(* CoDeSys 2.3.9.48 project: test.pro *)
(* Libraries: SysLibRtc.lib 8.11.10 11:37:48, SerComm.lib 31.5.11 08:06:48, C:\Stuff\Wago\libs\WagoLibDaylightSaving.lib 26.2.10 09:49:28, Building_common.lib 28.9.15 12:45:22, Standard.lib 8.11.10 11:37:48, C:\Stuff\Wago\libs\WagoBuilding_01.lib 21.3.16 16:30:58, WagoLibSSL.lib 25.2.13 12:47:14, SYSLIBCALLBACK.LIB 8.11.10 11:37:48, Ethernet.lib 8.11.10 11:37:48, C:\Stuff\Wago\libs\oscat_building_100.lib 2.1.18 20:06:49, C:\Stuff\Wago\libs\oscat_basic_333.lib 2.1.18 20:07:40 *)

(* PLC configuration (modules and I/O channels)
0750-1405 16 DI 24V DC 3.0ms [Type_1_16_Channels] node 0, in %IB0 out %QB0 {INTTypePAAssignment = PLC; INTTypeModule = plugged}
  in10 AT %IX0.0 [BOOLOnX_I] Ch_1 Digital input
  in11 AT %IX0.1 [BOOLOnX_I] Ch_2 Digital input
  in12 AT %IX0.2 [BOOLOnX_I] Ch_3 Digital input
  in13 AT %IX0.3 [BOOLOnX_I] Ch_4 Digital input
  in14 AT %IX0.4 [BOOLOnX_I] Ch_5 Digital input
  in15 AT %IX0.5 [BOOLOnX_I] Ch_6 Digital input
  in16 AT %IX0.6 [BOOLOnX_I] Ch_7 Digital input
  in17 AT %IX0.7 [BOOLOnX_I] Ch_8 Digital input
  in18 AT %IX0.8 [BOOLOnX_I] Ch_9 Digital input
  in19 AT %IX0.9 [BOOLOnX_I] Ch_10 Digital input
  in1A AT %IX0.10 [BOOLOnX_I] Ch_11 Digital input
  in1B AT %IX0.11 [BOOLOnX_I] Ch_12 Digital input
  in1C AT %IX0.12 [BOOLOnX_I] Ch_13 Digital input
  in1D AT %IX0.13 [BOOLOnX_I] Ch_14 Digital input
  in1E AT %IX0.14 [BOOLOnX_I] Ch_15 Digital input
  in1F AT %IX0.15 [BOOLOnX_I] Ch_16 Digital input
0750-0430 8 DI 24 V DC 3.0ms [Type_1_8_Channels] node 1, in %IB0 out %QB0 {INTTypePAAssignment = PLC; INTTypeModule = plugged}
  in20 AT %IX1.0 [BOOLOnX_I] Ch_1 Digital input
  in21 AT %IX1.1 [BOOLOnX_I] Ch_2 Digital input
  in22 AT %IX1.2 [BOOLOnX_I] Ch_3 Digital input
  in23 AT %IX1.3 [BOOLOnX_I] Ch_4 Digital input
  in24 AT %IX1.4 [BOOLOnX_I] Ch_5 Digital input
  in25 AT %IX1.5 [BOOLOnX_I] Ch_6 Digital input
  in26 AT %IX1.6 [BOOLOnX_I] Ch_7 Digital input
  in27 AT %IX1.7 [BOOLOnX_I] Ch_8 Digital input
0750-0430 8 DI 24 V DC 3.0ms [Type_1_8_Channels] node 2, in %IB2 out %QB0 {INTTypePAAssignment = PLC; INTTypeModule = plugged}
  in30 AT %IX1.8 [BOOLOnX_I] Ch_1 Digital input
  in31 AT %IX1.9 [BOOLOnX_I] Ch_2 Digital input
  in32 AT %IX1.10 [BOOLOnX_I] Ch_3 Digital input
  in33 AT %IX1.11 [BOOLOnX_I] Ch_4 Digital input
  in34 AT %IX1.12 [BOOLOnX_I] Ch_5 Digital input
  in35 AT %IX1.13 [BOOLOnX_I] Ch_6 Digital input
  in36 AT %IX1.14 [BOOLOnX_I] Ch_7 Digital input
  in37 AT %IX1.15 [BOOLOnX_I] Ch_8 Digital input
0750-0430 8 DI 24 V DC 3.0ms [Type_1_8_Channels] node 3, in %IB3 out %QB0 {INTTypePAAssignment = PLC; INTTypeModule = plugged}
  in40 AT %IX2.0 [BOOLOnX_I] Ch_1 Digital input
  in41 AT %IX2.1 [BOOLOnX_I] Ch_2 Digital input
  in42 AT %IX2.2 [BOOLOnX_I] Ch_3 Digital input
  in43 AT %IX2.3 [BOOLOnX_I] Ch_4 Digital input
  in44 AT %IX2.4 [BOOLOnX_I] Ch_5 Digital input
  in45 AT %IX2.5 [BOOLOnX_I] Ch_6 Digital input
  in46 AT %IX2.6 [BOOLOnX_I] Ch_7 Digital input
  in47 AT %IX2.7 [BOOLOnX_I] Ch_8 Digital input
0750-0402 4 DI 24 V DC 3.0ms [Type_1_4_Channels] node 4, in %IB4 out %QB0 {INTTypePAAssignment = PLC; INTTypeModule = plugged}
  in50 AT %IX2.8 [BOOLOnX_I] Ch_1 Digital input
  in51 AT %IX2.9 [BOOLOnX_I] Ch_2 Digital input
  in52 AT %IX2.10 [BOOLOnX_I] Ch_3 Digital input
  in53 AT %IX2.11 [BOOLOnX_I] Ch_4 Digital input
0750-0418 2 DI 24V DC 3.0ms / Diagnosis / Acknowledgement [Type_6_2_Channels] node 5, in %IB5 out %QB0 {INTTypePAAssignment = PLC; INTTypeModule = plugged}
  in60 AT %IX2.12 [BOOLOnX_I] Digital input
  in61 AT %IX2.13 [BOOLOnX_I] Digital input
  AT %IX2.14 [BOOLOnX_I] Diagnostic
  AT %IX2.15 [BOOLOnX_I] Diagnostic
  AT %QX0.2 [BOOLOnX_Q] Reset diagnostic
  AT %QX0.3 [BOOLOnX_Q] Reset diagnostic
0750-0418 2 DI 24V DC 3.0ms / Diagnosis / Acknowledgement [Type_6_2_Channels] node 6, in %IX2.12 out %QB0 {INTTypePAAssignment = PLC; INTTypeModule = plugged}
  in70 AT %IX3.0 [BOOLOnX_I] Digital input
  in71 AT %IX3.1 [BOOLOnX_I] Digital input
  AT %IX3.2 [BOOLOnX_I] Diagnostic
  AT %IX3.3 [BOOLOnX_I] Diagnostic
  AT %QX0.6 [BOOLOnX_Q] Reset diagnostic
  AT %QX0.7 [BOOLOnX_Q] Reset diagnostic
0750-0418 2 DI 24V DC 3.0ms / Diagnosis / Acknowledgement [Type_6_2_Channels] node 7, in %IB6 out %QX0.4 {INTTypePAAssignment = PLC; INTTypeModule = plugged}
  in80 AT %IX3.4 [BOOLOnX_I] Digital input
  in81 AT %IX3.5 [BOOLOnX_I] Digital input
  AT %IX3.6 [BOOLOnX_I] Diagnostic
  AT %IX3.7 [BOOLOnX_I] Diagnostic
  AT %QX0.10 [BOOLOnX_Q] Reset diagnostic
  AT %QX0.11 [BOOLOnX_Q] Reset diagnostic
0750-0418 2 DI 24V DC 3.0ms / Diagnosis / Acknowledgement [Type_6_2_Channels] node 8, in %IX3.4 out %QB1 {INTTypePAAssignment = PLC; INTTypeModule = plugged}
  in90 AT %IX3.8 [BOOLOnX_I] Digital input
  in91 AT %IX3.9 [BOOLOnX_I] Digital input
  AT %IX3.10 [BOOLOnX_I] Diagnostic
  AT %IX3.11 [BOOLOnX_I] Diagnostic
  AT %QX0.14 [BOOLOnX_Q] Reset diagnostic
  AT %QX0.15 [BOOLOnX_Q] Reset diagnostic
0750-0418 2 DI 24V DC 3.0ms / Diagnosis / Acknowledgement [Type_6_2_Channels] node 9, in %IB7 out %QX0.12 {INTTypePAAssignment = PLC; INTTypeModule = plugged}
  inA0 AT %IX3.12 [BOOLOnX_I] Digital input
  inA1 AT %IX3.13 [BOOLOnX_I] Digital input
  AT %IX3.14 [BOOLOnX_I] Diagnostic
  AT %IX3.15 [BOOLOnX_I] Diagnostic
  AT %QX1.2 [BOOLOnX_Q] Reset diagnostic
  AT %QX1.3 [BOOLOnX_Q] Reset diagnostic
0750-0418 2 DI 24V DC 3.0ms / Diagnosis / Acknowledgement [Type_6_2_Channels] node 10, in %IX3.12 out %QB2 {INTTypePAAssignment = PLC; INTTypeModule = plugged}
  inB0 AT %IX4.0 [BOOLOnX_I] Digital input
  inB1 AT %IX4.1 [BOOLOnX_I] Digital input
  AT %IX4.2 [BOOLOnX_I] Diagnostic
  AT %IX4.3 [BOOLOnX_I] Diagnostic
  AT %QX1.6 [BOOLOnX_Q] Reset diagnostic
  AT %QX1.7 [BOOLOnX_Q] Reset diagnostic
0750-0418 2 DI 24V DC 3.0ms / Diagnosis / Acknowledgement [Type_6_2_Channels] node 11, in %IB8 out %QX1.4 {INTTypePAAssignment = PLC; INTTypeModule = plugged}
  inC0 AT %IX4.4 [BOOLOnX_I] Digital input
  inC01 AT %IX4.5 [BOOLOnX_I] Digital input
  AT %IX4.6 [BOOLOnX_I] Diagnostic
  AT %IX4.7 [BOOLOnX_I] Diagnostic
  AT %QX1.10 [BOOLOnX_Q] Reset diagnostic
  AT %QX1.11 [BOOLOnX_Q] Reset diagnostic
0750-1504 16 DO 24V DC 0.5A [Type_10_16_Channels] node 12, in %IX4.4 out %QB3 {INTTypePAAssignment = PLC; INTTypeModule = plugged}
  out10 AT %QX1.12 [BOOLOnX_Q] Ch_1 Digital output
  out11 AT %QX1.13 [BOOLOnX_Q] Ch_2 Digital output
  out12 AT %QX1.14 [BOOLOnX_Q] Ch_3 Digital output
  out13 AT %QX1.15 [BOOLOnX_Q] Ch_4 Digital output
  out14 AT %QX2.0 [BOOLOnX_Q] Ch_5 Digital output
  out15 AT %QX2.1 [BOOLOnX_Q] Ch_6 Digital output
  out16 AT %QX2.2 [BOOLOnX_Q] Ch_7 Digital output
  out17 AT %QX2.3 [BOOLOnX_Q] Ch_8 Digital output
  out18 AT %QX2.4 [BOOLOnX_Q] Ch_9 Digital output
  out19 AT %QX2.5 [BOOLOnX_Q] Ch_10 Digital output
  out1A AT %QX2.6 [BOOLOnX_Q] Ch_11 Digital output
  out1B AT %QX2.7 [BOOLOnX_Q] Ch_12 Digital output
  out1C AT %QX2.8 [BOOLOnX_Q] Ch_13 Digital output
  out1D AT %QX2.9 [BOOLOnX_Q] Ch_14 Digital output
  out1E AT %QX2.10 [BOOLOnX_Q] Ch_15 Digital output
  out1F AT %QX2.11 [BOOLOnX_Q] Ch_16 Digital output
0750-1504 16 DO 24V DC 0.5A [Type_10_16_Channels] node 13, in %IB9 out %QX1.12 {INTTypePAAssignment = PLC; INTTypeModule = plugged}
  out20 AT %QX2.12 [BOOLOnX_Q] Ch_1 Digital output
  out21 AT %QX2.13 [BOOLOnX_Q] Ch_2 Digital output
  out22 AT %QX2.14 [BOOLOnX_Q] Ch_3 Digital output
  out23 AT %QX2.15 [BOOLOnX_Q] Ch_4 Digital output
  out24 AT %QX3.0 [BOOLOnX_Q] Ch_5 Digital output
  out25 AT %QX3.1 [BOOLOnX_Q] Ch_6 Digital output
  out26 AT %QX3.2 [BOOLOnX_Q] Ch_7 Digital output
  out27 AT %QX3.3 [BOOLOnX_Q] Ch_8 Digital output
  out28 AT %QX3.4 [BOOLOnX_Q] Ch_9 Digital output
  out29 AT %QX3.5 [BOOLOnX_Q] Ch_10 Digital output
  out2A AT %QX3.6 [BOOLOnX_Q] Ch_11 Digital output
  out2B AT %QX3.7 [BOOLOnX_Q] Ch_12 Digital output
  out2C AT %QX3.8 [BOOLOnX_Q] Ch_13 Digital output
  out2D AT %QX3.9 [BOOLOnX_Q] Ch_14 Digital output
  out2E AT %QX3.10 [BOOLOnX_Q] Ch_15 Digital output
  out2F AT %QX3.11 [BOOLOnX_Q] Ch_16 Digital output
0750-1504 16 DO 24V DC 0.5A [Type_10_16_Channels] node 14, in %IB9 out %QX2.12 {INTTypePAAssignment = PLC; INTTypeModule = plugged}
  out30 AT %QX3.12 [BOOLOnX_Q] Ch_1 Digital output
  out31 AT %QX3.13 [BOOLOnX_Q] Ch_2 Digital output
  out32 AT %QX3.14 [BOOLOnX_Q] Ch_3 Digital output
  out33 AT %QX3.15 [BOOLOnX_Q] Ch_4 Digital output
  out34 AT %QX4.0 [BOOLOnX_Q] Ch_5 Digital output
  out35 AT %QX4.1 [BOOLOnX_Q] Ch_6 Digital output
  out36 AT %QX4.2 [BOOLOnX_Q] Ch_7 Digital output
  out37 AT %QX4.3 [BOOLOnX_Q] Ch_8 Digital output
  out38 AT %QX4.4 [BOOLOnX_Q] Ch_9 Digital output
  out39 AT %QX4.5 [BOOLOnX_Q] Ch_10 Digital output
  out3A AT %QX4.6 [BOOLOnX_Q] Ch_11 Digital output
  out3B AT %QX4.7 [BOOLOnX_Q] Ch_12 Digital output
  out3C AT %QX4.8 [BOOLOnX_Q] Ch_13 Digital output
  out3D AT %QX4.9 [BOOLOnX_Q] Ch_14 Digital output
  out3E AT %QX4.10 [BOOLOnX_Q] Ch_15 Digital output
  out3F AT %QX4.11 [BOOLOnX_Q] Ch_16 Digital output
0750-0517 2 DO 230V AC 1.0A Rel 2CO (PotFree) [Type_10_2_Channels] node 15, in %IB9 out %QX3.12 {INTTypePAAssignment = PLC; INTTypeModule = plugged}
  out40 AT %QX4.12 [BOOLOnX_Q] Ch_1 Digital output
  out41 AT %QX4.13 [BOOLOnX_Q] Ch_2 Digital output
0750-0517 2 DO 230V AC 1.0A Rel 2CO (PotFree) [Type_10_2_Channels] node 16, in %IB9 out %QX4.12 {INTTypePAAssignment = PLC; INTTypeModule = plugged}
  out50 AT %QX4.14 [BOOLOnX_Q] Ch_1 Digital output
  out51 AT %QX4.15 [BOOLOnX_Q] Ch_2 Digital output
0750-0517 2 DO 230V AC 1.0A Rel 2CO (PotFree) [Type_10_2_Channels] node 17, in %IB9 out %QX4.14 {INTTypePAAssignment = PLC; INTTypeModule = plugged}
  out60 AT %QX5.0 [BOOLOnX_Q] Ch_1 Digital output
  out61 AT %QX5.1 [BOOLOnX_Q] Ch_2 Digital output
0750-0517 2 DO 230V AC 1.0A Rel 2CO (PotFree) [Type_10_2_Channels] node 18, in %IB9 out %QB10 {INTTypePAAssignment = PLC; INTTypeModule = plugged}
  out70 AT %QX5.2 [BOOLOnX_Q] Ch_1 Digital output
  out71 AT %QX5.3 [BOOLOnX_Q] Ch_2 Digital output
0750-0513 2 DO 250V AC 2.0A Rel 2NO (PotFree) [Type_10_2_Channels] node 19, in %IB9 out %QX5.2 {INTTypePAAssignment = PLC; INTTypeModule = plugged}
  out80 AT %QX5.4 [BOOLOnX_Q] Ch_1 Digital output
  out81 AT %QX5.5 [BOOLOnX_Q] Ch_2 Digital output
AT %IX4.8 [BOOLOnX_I] Channel 1 Diagnostic bit 0
AT %IX4.9 [BOOLOnX_I] Channel 1 Diagnostic bit 1
AT %IX4.10 [BOOLOnX_I] Channel 2 Diagnostic bit 0
AT %IX4.11 [BOOLOnX_I] Channel 2 Diagnostic bit 1
out90 AT %QX5.6 [BOOLOnX_Q] Digital output 1
out91 AT %QX5.7 [BOOLOnX_Q] Digital output 2
AT %IX4.12 [BOOLOnX_I] Channel 1 Diagnostic bit 0
AT %IX4.13 [BOOLOnX_I] Channel 1 Diagnostic bit 1
AT %IX4.14 [BOOLOnX_I] Channel 2 Diagnostic bit 0
AT %IX4.15 [BOOLOnX_I] Channel 2 Diagnostic bit 1
outA0 AT %QX5.10 [BOOLOnX_Q] Digital output 1
out1A1 AT %QX5.11 [BOOLOnX_Q] Digital output 2
AT %IX5.0 [BOOLOnX_I] Channel 1 Diagnostic bit 0
AT %IX5.1 [BOOLOnX_I] Channel 1 Diagnostic bit 1
AT %IX5.2 [BOOLOnX_I] Channel 2 Diagnostic bit 0
AT %IX5.3 [BOOLOnX_I] Channel 2 Diagnostic bit 1
outB0 AT %QX5.14 [BOOLOnX_Q] Digital output 1
outB1 AT %QX5.15 [BOOLOnX_Q] Digital output 2
Fieldbus variables [FB_VARS] node 1, in %IB0 out %QB0
Flag variables [FLAG_VARS] node 2, in %IB0 out %QB0
Modbus-Master [MB_MASTER] node 3, in %IB0 out %QB0
*)

(* Task configuration *)
TASK MainTask (PRIORITY := 1); (* freewheeling *)
	PLC_PRG();
END_TASK
TASK UpdateClock (PRIORITY := 3, INTERVAL := T#1000ms);
	ReadClock();
END_TASK

(* POU PLC_PRG, ST *)
PROGRAM PLC_PRG
VAR
	pompaCWU:FbLatchedRelay;
	pompaCWUVis:BOOL;
	pompaCWUTOF:TOF;
	pompaCWUTOFTRIG:F_TRIG;

	tvSat:FbLatchedRelay;
	tvSatVis:BOOL;
	tvSatTOF:TOF;
	tvSatTOFTRIG:F_TRIG;
END_VAR
Swiatlo;
SterowanieRolet;

pompaCWU(xButton:=(LazienkaPietro.Swiatlo OR LazienkaParter.Swiatlo OR KuchniaJadalnia.Swiatlo OR pompaCWUVis), xCentralOff:=pompaCWUTOFTRIG.Q);
pompaCWUTOF(IN:=LazienkaPietro.swLazienkaD.xActuator,PT:=T#10M);
pompaCWUTOFTRIG(CLK:=pompaCWUTOF.Q);
out2C:=pompaCWU.xActuator;

(*TODOultimate off*)

(*TVSAT off*)
END_PROGRAM

(* POU Swiatlo, ST *)
PROGRAM Swiatlo
VAR

END_VAR
GarazKotlownia;
GarderobaStrych;
Korytarz;
KuchniaJadalnia;
LazienkaParter;
LazienkaPietro;
PokojPolnoc;
PokojPoludnie;
Salon;
Sypialnia;
WiatrolapSpizarnia;
END_PROGRAM

(* POU Swiatlo2/GarazKotlownia, ST *)
PROGRAM GarazKotlownia
VAR
	swGarazDrzwiKotlowni : BOOL;
	visGaraz : BOOL;
	swGarazBrama: BOOL;
	swGarazBiurko: BOOL;
	garazTOF:TOF;
	garazTOFTRIG:F_TRIG;
	garazClicker: CLICK;
	wlaczWszystkieSw: BOOL := FALSE;
	wylaczWszystkieSw: BOOL := FALSE;
	visKotlownia: BOOL;
	kotlowniaTOF:TOF;
	kotlowniaTOFTRIG:F_TRIG;
	kotlowniaClicker: FbWB_EvaluateMultipleClicks;
	garaz:SwiatloOpFUN;
END_VAR
VAR RETAIN
	swGaraz: FbLatchedRelay;
	swKotlownia: FbLatchedRelay;
END_VAR
(*----------Garaz--------*)
(*swGaraz(xButton:= (garazClicker.single OR garazClicker.double OR visGaraz), xCentralOn:=wlaczWszystkieSw, xCentralOff:=garazTOFTRIG.Q);
out10:=swGaraz.xActuator;
garazTOF(IN:=garazClicker.single, PT:=T#2M);
garazTOFTRIG(CLK:=garazTOF.Q);
garazClicker(in:=(in10 OR in20));*)

garaz(wejscieSterujace:=(in10),wlaczWszystkie:=wlaczWszystkieSw,wylaczWszystkie:=wylaczWszystkieSw,sterowanieVis:=visGaraz);
out10:=garaz.wyjscie;

(*----------Kotlownia-------*)
swKotlownia(xButton:=(kotlowniaClicker.xMultipleClick OR kotlowniaClicker.xFewerClick OR visKotlownia), xCentralOn:=wlaczWszystkieSw, xCentralOff:=kotlowniaTOFTRIG.Q);
kotlowniaTOF(IN:=kotlowniaClicker.xFewerClick,PT:=T#5M);
kotlowniaTOFTRIG(CLK:=kotlowniaTOF.Q);
kotlowniaClicker(xButton:=(in11 OR in21));
out11:=swKotlownia.xActuator;
out90:=garaz.wyjscie;
out91:=garaz.wyjscie;
outA0:=garaz.wyjscie;
out1A1:=garaz.wyjscie;
outB0:=garaz.wyjscie;
outB1:=garaz.wyjscie;
END_PROGRAM

(* POU Swiatlo2/SwiatloOpFUN, ST *)
FUNCTION_BLOCK SwiatloOpFUN
VAR_INPUT
	wejscieSterujace :BOOL;
	wlaczWszystkie:BOOL;
	wylaczWszystkie:BOOL;
	sterowanieVis:BOOL;
END_VAR
VAR_OUTPUT
	wyjscie :BOOL;
END_VAR
VAR
	przelacznik:FbLatchedRelay;
	opoznienieTOF:TOF;
	opoznienieTOFTRIG:F_TRIG;
	clicker:Fb_Click;
END_VAR
przelacznik(xButton:=(clicker.xSingle OR clicker.xDouble OR  sterowanieVis), xCentralOn:=wlaczWszystkie, xCentralOff:=(opoznienieTOFTRIG.Q OR wylaczWszystkie));
opoznienieTOF(IN:=clicker.xSingle, PT:=T#3m);
opoznienieTOFTRIG(CLK:=opoznienieTOF.Q);
clicker(xSwitch:=wejscieSterujace,uiT_10tel_s:=5);
wyjscie:=przelacznik.xActuator;
END_FUNCTION_BLOCK

(* POU Swiatlo2/GarderobaStrych, ST *)
PROGRAM GarderobaStrych
VAR
	swStrych: FbLatchedRelay;
	visStrych: BOOL;
	strychTOF:TOF;
	strychTOFTRIG:F_TRIG;
	strychClicker: FbWB_EvaluateMultipleClicks;
	swSchowekPietro: FbLatchedRelay;
	visSchowekPietro: BOOL;
	schowekPietroTOF:TOF;
	schowekPietroTOFTRIG:F_TRIG;
	schowekPietroClicker: FbWB_EvaluateMultipleClicks;
	wlaczWszystkieSw: BOOL:=FALSE;
	wylaczWszystkieSw: BOOL:=FALSE;
END_VAR
swSchowekPietro(xButton:=(schowekPietroClicker.xMultipleClick OR schowekPietroClicker.xFewerClick OR visSchowekPietro),xCentralOn:=wlaczWszystkieSw,xCentralOff:=schowekPietroTOFTRIG.Q);
out25:=swSchowekPietro.xActuator;
schowekPietroTOF(IN:=schowekPietroClicker.xFewerClick,PT:=T#2m);
schowekPietroTOFTRIG(CLK:=schowekPietroTOF.Q);
schowekPietroClicker(xButton:=in34,bNumberOfClicks:=2);

swStrych(xButton:=(strychClicker.xMultipleClick OR strychTOFTRIG.Q OR visStrych), xCentralOn:=wlaczWszystkieSw,xCentralOff:=strychTOFTRIG.Q);
out26:=swStrych.xActuator;
strychTOF(IN:=strychClicker.xFewerClick,PT:=T#10m);
strychTOFTRIG(CLK:=strychTOF.Q);
strychClicker(xButton:=in35,bNumberOfClicks:=2);
END_PROGRAM

(* POU Swiatlo2/Korytarz, ST *)
PROGRAM Korytarz
VAR
	swKorytarz: FbLatchedRelay;
	visKorytarz: BOOL;
	swKorytarzPietro: FbLatchedRelay;
	visKorytarzPietro: BOOL;
	wlaczWszystkieSw: BOOL:=FALSE;
	wylaczWszystkieSw: BOOL:=FALSE;
END_VAR
swKorytarz(xButton:=(in1D OR visKorytarz), xCentralOn:=wlaczWszystkieSw, xCentralOff:=wylaczWszystkieSw);
out1D:=swKorytarz.xActuator;

swKorytarzPietro(xButton:=(in1F OR visKorytarzPietro), xCentralOn:=wlaczWszystkieSw, xCentralOff:=wylaczWszystkieSw);
out1F:=swKorytarzPietro.xActuator;
END_PROGRAM

(* POU Swiatlo2/KuchniaJadalnia, ST *)
PROGRAM KuchniaJadalnia
VAR
	swJadalnia: FbLatchedRelay;
	visJadalnia: BOOL;
	swBlat: FbLatchedRelay;
	visBlat: BOOL;
	swMeble: FbLatchedRelay;
	visMeble: BOOL;
	wlaczWszystkieSw: BOOL:=FALSE;
	wylaczWszystkieSw: BOOL:=FALSE;
	swSufit: FbLatchedRelay;
	visSufit: BOOL;
	swiatlo:BOOL;
END_VAR
(*----------Kuchnia--------------*)
swBlat(xButton:=(in17 OR visBlat), xCentralOn:=wlaczWszystkieSw,  xCentralOff:=wylaczWszystkieSw);
out16:=swBlat.xActuator;
swMeble(xButton:=(in16 OR visMeble), xCentralOn:=wlaczWszystkieSw,  xCentralOff:=wylaczWszystkieSw);
out17:=swMeble.xActuator;
swSufit(xButton:=(in16 OR visSufit), xCentralOn:=wlaczWszystkieSw,  xCentralOff:=wylaczWszystkieSw);
out1E:=swSufit.xActuator;

(*----------Jadalnia--------------*)
swJadalnia(xButton:=(in18 OR visJadalnia), xCentralOn:=wlaczWszystkieSw,xCentralOff:=wylaczWszystkieSw);
out18:=swJadalnia.xActuator;

Swiatlo:=swBlat.xActuator OR swMeble.xActuator OR swSufit.xActuator;
END_PROGRAM

(* POU Swiatlo2/LazienkaParter, ST *)
PROGRAM LazienkaParter
VAR
	visMalaLazienkaPrysznic:BOOL;
	swMalaLazienkaLustro: FbLatchedRelay;
	visMalaLazienkaLustro: BOOL;
	swMalaLazienka: FbLatchedRelay;
	visMalaLazienka: BOOL;
	swMalaLazienkaPrysznic: FbLatchedRelay;
	wlaczWszystkieSw: BOOL:=FALSE;
	wylaczWszystkieSw: BOOL:=FALSE;
	swiatlo: BOOL;
END_VAR
(*---------Mala lazienka -------*)
swMalaLazienka(xButton:=(in13 OR visMalaLazienka), xCentralOn:=wlaczWszystkieSw, xCentralOff:=wylaczWszystkieSw);
out13:=swMalaLazienka.xActuator;
swMalaLazienkaPrysznic(xButton:=(in14 OR in24 OR visMalaLazienkaPrysznic), xCentralOn:=wlaczWszystkieSw, xCentralOff:=wylaczWszystkieSw);
out50:=swMalaLazienkaPrysznic.xActuator;
swMalaLazienkaLustro(xButton:=(in15 OR in25 OR visMalaLazienkaLustro), xCentralOn:=wlaczWszystkieSw,xCentralOff:=wylaczWszystkieSw);
out15:=swMalaLazienkaLustro.xActuator;

Swiatlo:=swMalaLazienka.xActuator OR swMalaLazienkaPrysznic.xActuator OR swMalaLazienkaLustro.xActuator;
END_PROGRAM

(* POU Swiatlo2/LazienkaPietro, ST *)
PROGRAM LazienkaPietro
VAR
	swLustroLD: FbLatchedRelay;
	visLustroLD: BOOL;
	swLazienkaD: FbLatchedRelay;
	visLazienkaD: BOOL;
	swBlatLD: FbLatchedRelay;
	visBlatLD: BOOL;
	swPrysznicLD: FbLatchedRelay;
	visPrysznicLD: BOOL;

	swLazienkaLedTrigger: R_TRIG;
	visLedLD: BOOL;
	wlaczWszystkieSw: BOOL:=FALSE;
	wylaczWszystkieSw: BOOL:=FALSE;
	swiatlo:BOOL;
END_VAR
(*----------------Duza lazienka------------*)
swLustroLD(xButton:=(in36 OR visLustroLD), xCentralOn:=wlaczWszystkieSw,xCentralOff:=wylaczWszystkieSw);
out27:=swLustroLD.xActuator;
swLazienkaD(xButton:=(in37 OR visLazienkaD), xCentralOn:=wlaczWszystkieSw,xCentralOff:=wylaczWszystkieSw);
out28:=swLazienkaD.xActuator;
swBlatLD(xButton:=(in40 OR visBlatLD), xCentralOn:=wlaczWszystkieSw,xCentralOff:=wylaczWszystkieSw);
out40:=swBlatLD.xActuator;
swPrysznicLD(xButton:=(in41 OR visPrysznicLD), xCentralOn:=wlaczWszystkieSw,xCentralOff:=wylaczWszystkieSw);
out41:=swPrysznicLD.xActuator;

swLazienkaLedTrigger(CLK:=(in43 OR visLedLD));
IF swLazienkaLedTrigger.Q THEN
	IF NOT (out29 OR out2A) THEN
		visBlatLD := visPrysznicLD := TRUE;
	ELSE
		visBlatLD := visPrysznicLD := FALSE;
	END_IF;
END_IF;

Swiatlo:=swLazienkaD.xActuator OR swLustroLD.xActuator OR swBlatLD.xActuator OR swPrysznicLD.xActuator;
END_PROGRAM

(* POU Swiatlo2/PokojPolnoc, ST *)
PROGRAM PokojPolnoc
VAR
	swPokojPolnoc: FbLatchedRelay;
	visPokojPolnoc: BOOL;
	wlaczWszystkieSw: BOOL:=FALSE;
	wylaczWszystkieSw: BOOL:=FALSE;
END_VAR
swPokojPolnoc(xButton:=(in33 OR visPokojPolnoc),xCentralOn:=wlaczWszystkieSw,xCentralOff:=wylaczWszystkieSw);
out24:=swPokojPolnoc.xActuator;
END_PROGRAM

(* POU Swiatlo2/PokojPoludnie, ST *)
PROGRAM PokojPoludnie
VAR
	swPokojPoludnie: FbLatchedRelay;
	visPokojPoludnie: BOOL;
	wlaczWszystkieSw: BOOL:=FALSE;
	wylaczWszystkieSw: BOOL:=FALSE;
END_VAR
swPokojPoludnie(xButton:=(in32 OR visPokojPoludnie), xCentralOn:=wlaczWszystkieSw,xCentralOff:=wylaczWszystkieSw);
out23:=swPokojPoludnie.xActuator;
END_PROGRAM

(* POU Swiatlo2/Salon, ST *)
PROGRAM Salon
VAR
	swSalonCentralne: FbLatchedRelay;
	visSalonCentralne: BOOL;
	swSalonSciana: FbLatchedRelay;
	visSalonSciana: BOOL;
	swSalonKinkiet: FbLatchedRelay;
	visSalonKinkiet: BOOL;
	swSalonSufit: FbLatchedRelay;
	visSalonSufit: BOOL;
	wlaczWszystkieSw: BOOL:=FALSE;
	wylaczWszystkieSw: BOOL:=FALSE;
END_VAR
(*----------Salon-----------------*)
swSalonCentralne(xButton:=(in19 OR visSalonCentralne), xCentralOn:=wlaczWszystkieSw, xCentralOff:=wylaczWszystkieSw);
out19:=swSalonCentralne.xActuator;
swSalonSciana(xButton:=(in1A OR visSalonSciana), xCentralOn:=wlaczWszystkieSw, xCentralOff:=wylaczWszystkieSw);
out1A:=swSalonSciana.xActuator;
swSalonKinkiet(xButton:=(in1B OR visSalonKinkiet), xCentralOn:=wlaczWszystkieSw, xCentralOff:=wylaczWszystkieSw);
out1B:=swSalonKinkiet.xActuator;
swSalonSufit(xButton:=(in1C OR visSalonSufit), xCentralOn:=wlaczWszystkieSw, xCentralOff:=wylaczWszystkieSw);
out1C:=swSalonSufit.xActuator;
END_PROGRAM

(* POU Swiatlo2/Sypialnia, ST *)
PROGRAM Sypialnia
VAR
	swSypialniaLozko: FbLatchedRelay;
	visSypialniaLozko: BOOL;
	swSypialnia: FbLatchedRelay;
	visSypialnia: BOOL;
	wlaczWszystkieSw: BOOL:=FALSE;
	wylaczWszystkieSw: BOOL:=FALSE;
END_VAR
swSypialniaLozko(xButton:=(in26 OR visSypialniaLozko), xCentralOn:=wlaczWszystkieSw, xCentralOff:=wylaczWszystkieSw);
out20:=swSypialniaLozko.xActuator;

swSypialnia(xButton:=(in27 OR visSypialnia), xCentralOn:=wlaczWszystkieSw, xCentralOff:=wylaczWszystkieSw);
out21:=swSypialnia.xActuator;
END_PROGRAM

(* POU Swiatlo2/WiatrolapSpizarnia, ST *)
PROGRAM WiatrolapSpizarnia
VAR
	swWiatrolap:FbLatchedRelay;
	visWiatrolap:BOOL;
	wiatrolapTOF:TOF;
	wiatrolapTOFTRIG:F_TRIG;
	wiatrolapClicker:CLICK;
	wlaczWszystkieSw: BOOL:=FALSE;
	wylaczWszystkieSw: BOOL:=FALSE;
	swSpizarnia:SwiatloOpFUN;
	visSpizarnia:BOOL;
END_VAR
(*---------Wiatrolap--------*)
swWiatrolap(xButton:=(in12), xCentralOn:=wlaczWszystkieSw, xCentralOff:=wiatrolapTOFTRIG.Q);
wiatrolapTOF(IN:=wiatrolapClicker.single, PT:=T#5m);
wiatrolapTOFTRIG(CLK:=wiatrolapTOF.Q);
wiatrolapClicker(in:=in12);
out12:=swWiatrolap.xActuator;

(*-----Spizarnia---------*)
swSpizarnia(wejscieSterujace:=in1E,
	wlaczWszystkie:=wlaczWszystkieSw,
	wylaczWszystkie:=wylaczWszystkieSw,
	sterowanieVis:=visSpizarnia);
out14:=swSpizarnia.wyjscie;
END_PROGRAM

(* POU Rolety2/SterowanieRolet, ST *)
PROGRAM SterowanieRolet
VAR
	kotlownia: RoletyFUN;
	kotlowniaUpVis: BOOL;
	kotlowniaDnVis: BOOL;
	kotlowniaLamelkiVis: BOOL;

	witrynaP:RoletyFUN;
	witrynaL:RoletyFUN;
	witrynaUpVis:BOOL;
	witrynaDnVis:BOOL;
	witrynaLamelkiVis:BOOL;

	salonWyjscie: RoletyFUN;
	salonWyjscieUpVis:BOOL;
	salonWyjscieDnVis:BOOL;
	salonWyjscieLamelkiVis:BOOL;

	jadalniaWyjscie: RoletyFUN;
	jadalniaWyjscieUpVis:BOOL;
	jadalniaWyjscieDnVis:BOOL;
	jadalniaWyjscieLamelkiVis:BOOL;

	jadalniaWitryna: RoletyFUN;
	jadalniaWitrynaUpVis:BOOL;
	jadalniaWitrynaDnVis:BOOL;
	jadalniaWitrynaLamelkiVis:BOOL;

	kuchnia: RoletyFUN;
	kuchniaUpVis:BOOL;
	kuchniaDnVis:BOOL;
	kuchniaLamelkiVis:BOOL;

	lazienkaParterR: RoletyFUN;
	lazienkaParterUpVis:BOOL;
	lazienkaParterDnVis:BOOL;
	lazienkaParterLamelkiVis:BOOL;

	lazienkaPietroR: RoletyFUN;
	lazienkaPietroUpVis:BOOL;
	lazienkaPietroDnVis:BOOL;
	lazienkaPietroLamelkiVis:BOOL;

	pokojPolnocR: RoletyFUN;
	pokojPolnocUpVis:BOOL;
	pokojPolnocDnVis:BOOL;
	pokojPolnocLamelkiVis:BOOL;

	pokojPoludnieR: RoletyFUN;
	pokojPoludnieUpVis:BOOL;
	pokojPoludnieDnVis:BOOL;
	pokojPoludnieLamelkiVis:BOOL;

	sypialniaR: RoletyFUN;
	sypialniaUpVis:BOOL;
	sypialniaDnVis:BOOL;
	sypialniaLamelkiVis:BOOL;

	sypialniaBalkonR: RoletyFUN;
	sypialniaBalkonUpVis:BOOL;
	sypialniaBalkonDnVis:BOOL;
	sypialniaBalkonLamelkiVis:BOOL;

	zamykanieWszystkieVis: BOOL;
	otwieranieWszystkieVis: BOOL;
	podniesStrefeDzienna:BOOL;
	opuscStrefeDzienna:BOOL;
	podniesPietro:BOOL;
	opuscPietro:BOOL;
       roletyParter : Fb_ShortLong:=(uiTS_10tel_s:=1, uiTL_10tel_s:=1, uiT_10tel_s :=5);
	roletyPietro : Fb_ShortLong:=(uiTS_10tel_s:=1, uiTL_10tel_s:=1, uiT_10tel_s :=5);
	roletyParterPoludnie:Fb_ShortLong:=(uiTS_10tel_s:=1, uiTL_10tel_s:=1, uiT_10tel_s :=5);
	roletyParterPolnoc:Fb_ShortLong:=(uiTS_10tel_s:=1, uiTL_10tel_s:=1, uiT_10tel_s :=5);
	opuscParterPoludnie:BOOL;
	podniesParterPoludnie:BOOL;
	opuscParterPolnoc:BOOL;
	podniesParterPolnoc:BOOL;
END_VAR
roletyParter(xSwitch:=inC0);
roletyPietro(xSwitch:=inC01);
roletyParterPoludnie(xSwitch:=in20);
roletyParterPolnoc(xSwitch:=in23);
podniesStrefeDzienna:=roletyParter.xShort;
opuscStrefeDzienna:=roletyParter.xLong;
podniesPietro:=roletyPietro.xShort;
opuscPietro:=roletyPietro.xLong;
opuscParterPoludnie:=roletyParterPoludnie.xLong;
podniesParterPoludnie:=roletyParterPoludnie.xShort;
opuscParterPolnoc:=roletyParterPolnoc.xLong;
podniesParterPolnoc:=roletyParterPolnoc.xShort;

kotlownia(wejscieSterujace:=in60,
		ZmiennaPodnoszenieVis:=kotlowniaUpVis,
		ZmiennaOpuszczanieVis:=kotlowniaDnVis,
		ZmiennaLamelkiVis:=kotlowniaLamelkiVis,
		PozycjaLameli:=10,
		CzasOtwarcia:=T#15s,
		CzasZamkniecia:=T#13s,
		MaxCzasDzialania:=T#20s,
		ZamykanieWszystkieVis:=zamykanieWszystkieVis,
		OtwieranieWszystkieVis:=otwieranieWszystkieVis);
out51:=kotlownia.WyjsciePodnoszenie;
out60:=kotlownia.WyjscieOpuszczanie;

witrynaP(wejscieSterujace:=in61,
		ZmiennaPodnoszenieVis:=witrynaUpVis,
		ZmiennaOpuszczanieVis:=witrynaDnVis,
		ZmiennaLamelkiVis:=witrynaLamelkiVis,
		PozycjaLameli:=10,
		CzasOtwarcia:=T#30s,
		CzasZamkniecia:=T#25s,
		MaxCzasDzialania:=T#30s,
		ZamykanieWszystkieVis:=zamykanieWszystkieVis OR opuscStrefeDzienna OR opuscParterPoludnie,
		OtwieranieWszystkieVis:=otwieranieWszystkieVis OR podniesStrefeDzienna OR podniesParterPoludnie);
out61:=witrynaP.WyjsciePodnoszenie;
out70:=witrynaP.WyjscieOpuszczanie;

witrynaL(wejscieSterujace:=in61,
		ZmiennaPodnoszenieVis:=witrynaUpVis,
		ZmiennaOpuszczanieVis:=witrynaDnVis,
		ZmiennaLamelkiVis:=witrynaLamelkiVis,
		PozycjaLameli:=10,
		CzasOtwarcia:=T#30s,
		CzasZamkniecia:=T#25s,
		MaxCzasDzialania:=T#30s,
		ZamykanieWszystkieVis:=zamykanieWszystkieVis OR opuscStrefeDzienna OR opuscParterPoludnie,
		OtwieranieWszystkieVis:=otwieranieWszystkieVis OR podniesStrefeDzienna OR podniesParterPoludnie);
out71:=witrynaL.WyjsciePodnoszenie;
out80:=witrynaL.WyjscieOpuszczanie;

salonWyjscie(wejscieSterujace:=in70,
		ZmiennaPodnoszenieVis:=salonWyjscieUpVis,
		ZmiennaOpuszczanieVis:=salonWyjscieDnVis,
		ZmiennaLamelkiVis:=salonWyjscieLamelkiVis,
		PozycjaLameli:=10,
		CzasOtwarcia:=T#30s,
		CzasZamkniecia:=T#25s,
		MaxCzasDzialania:=T#30s,
		ZamykanieWszystkieVis:=zamykanieWszystkieVis OR opuscStrefeDzienna OR opuscParterPoludnie,
		OtwieranieWszystkieVis:=otwieranieWszystkieVis OR podniesStrefeDzienna OR podniesParterPoludnie);
out31:=salonWyjscie.WyjsciePodnoszenie;
out32:=salonWyjscie.WyjscieOpuszczanie;

jadalniaWyjscie(wejscieSterujace:=in71,
		ZmiennaPodnoszenieVis:=jadalniaWyjscieUpVis,
		ZmiennaOpuszczanieVis:=jadalniaWyjscieDnVis,
		ZmiennaLamelkiVis:=jadalniaWyjscieLamelkiVis,
		PozycjaLameli:=10,
		CzasOtwarcia:=T#30s,
		CzasZamkniecia:=T#25s,
		MaxCzasDzialania:=T#30s,
		ZamykanieWszystkieVis:=zamykanieWszystkieVis OR opuscStrefeDzienna OR opuscParterPolnoc,
		OtwieranieWszystkieVis:=otwieranieWszystkieVis OR podniesStrefeDzienna OR podniesParterPolnoc);
out33:=jadalniaWyjscie.WyjsciePodnoszenie;
out34:=jadalniaWyjscie.WyjscieOpuszczanie;

jadalniaWitryna(wejscieSterujace:=in80,
		ZmiennaPodnoszenieVis:=jadalniaWitrynaUpVis,
		ZmiennaOpuszczanieVis:=jadalniaWitrynaDnVis,
		ZmiennaLamelkiVis:=jadalniaWitrynaLamelkiVis,
		PozycjaLameli:=10,
		CzasOtwarcia:=T#30s,
		CzasZamkniecia:=T#25s,
		MaxCzasDzialania:=T#30s,
		ZamykanieWszystkieVis:=zamykanieWszystkieVis OR opuscStrefeDzienna OR opuscParterPolnoc,
		OtwieranieWszystkieVis:=otwieranieWszystkieVis OR podniesStrefeDzienna OR podniesParterPolnoc);
out3F:=jadalniaWitryna.WyjsciePodnoszenie;
out2D:=jadalniaWitryna.WyjscieOpuszczanie;

kuchnia(wejscieSterujace:=in81,
		ZmiennaPodnoszenieVis:=kuchniaUpVis,
		ZmiennaOpuszczanieVis:=kuchniaDnVis,
		ZmiennaLamelkiVis:=kuchniaLamelkiVis,
		PozycjaLameli:=10,
		CzasOtwarcia:=T#30s,
		CzasZamkniecia:=T#25s,
		MaxCzasDzialania:=T#30s,
		ZamykanieWszystkieVis:=zamykanieWszystkieVis OR opuscStrefeDzienna OR opuscParterPolnoc,
		OtwieranieWszystkieVis:=otwieranieWszystkieVis OR podniesStrefeDzienna OR podniesParterPolnoc);
out2E:=kuchnia.WyjsciePodnoszenie;
out2F:=kuchnia.WyjscieOpuszczanie;

lazienkaParterR(wejscieSterujace:=in90,
		ZmiennaPodnoszenieVis:=lazienkaParterUpVis,
		ZmiennaOpuszczanieVis:=lazienkaParterDnVis,
		ZmiennaLamelkiVis:=lazienkaParterLamelkiVis,
		PozycjaLameli:=10,
		CzasOtwarcia:=T#10s,
		CzasZamkniecia:=T#9s,
		MaxCzasDzialania:=T#15s,
		ZamykanieWszystkieVis:=zamykanieWszystkieVis OR opuscStrefeDzienna,
		OtwieranieWszystkieVis:=otwieranieWszystkieVis OR podniesStrefeDzienna);
out35:=lazienkaParterR.WyjsciePodnoszenie;
out36:=lazienkaParterR.WyjscieOpuszczanie;

lazienkaPietroR(wejscieSterujace:=in91,
		ZmiennaPodnoszenieVis:=lazienkaPietroUpVis,
		ZmiennaOpuszczanieVis:=lazienkaPietroDnVis,
		ZmiennaLamelkiVis:=lazienkaPietroLamelkiVis,
		PozycjaLameli:=10,
		CzasOtwarcia:=T#20s,
		CzasZamkniecia:=T#17s,
		MaxCzasDzialania:=T#20s,
		ZamykanieWszystkieVis:=zamykanieWszystkieVis OR opuscPietro,
		OtwieranieWszystkieVis:=otwieranieWszystkieVis OR podniesPietro);
out37:=lazienkaPietroR.WyjsciePodnoszenie;
out38:=lazienkaPietroR.WyjscieOpuszczanie;

pokojPolnocR(wejscieSterujace:=inA0,
		ZmiennaPodnoszenieVis:=pokojPolnocUpVis,
		ZmiennaOpuszczanieVis:=pokojPolnocDnVis,
		ZmiennaLamelkiVis:=pokojPolnocLamelkiVis,
		PozycjaLameli:=10,
		CzasOtwarcia:=T#29s,
		CzasZamkniecia:=T#24s,
		MaxCzasDzialania:=T#29s,
		ZamykanieWszystkieVis:=zamykanieWszystkieVis OR opuscPietro,
		OtwieranieWszystkieVis:=otwieranieWszystkieVis OR podniesPietro);
out81:=pokojPolnocR.WyjsciePodnoszenie;
out30:=pokojPolnocR.WyjscieOpuszczanie;

pokojPoludnieR(wejscieSterujace:=inA1,
		ZmiennaPodnoszenieVis:=pokojPoludnieUpVis,
		ZmiennaOpuszczanieVis:=pokojPoludnieDnVis,
		ZmiennaLamelkiVis:=pokojPoludnieLamelkiVis,
		PozycjaLameli:=10,
		CzasOtwarcia:=T#29s,
		CzasZamkniecia:=T#24s,
		MaxCzasDzialania:=T#29s,
		ZamykanieWszystkieVis:=zamykanieWszystkieVis OR opuscPietro,
		OtwieranieWszystkieVis:=otwieranieWszystkieVis OR podniesPietro);
out39:=pokojPoludnieR.WyjsciePodnoszenie;
out3A:=pokojPoludnieR.WyjscieOpuszczanie;

sypialniaR(wejscieSterujace:=inB0,
		ZmiennaPodnoszenieVis:=sypialniaUpVis,
		ZmiennaOpuszczanieVis:=sypialniaDnVis,
		ZmiennaLamelkiVis:=sypialniaLamelkiVis,
		PozycjaLameli:=10,
		CzasOtwarcia:=T#20s,
		CzasZamkniecia:=T#17s,
		MaxCzasDzialania:=T#20s,
		ZamykanieWszystkieVis:=zamykanieWszystkieVis OR opuscPietro,
		OtwieranieWszystkieVis:=otwieranieWszystkieVis  OR podniesPietro);
out3B:=sypialniaR.WyjsciePodnoszenie;
out3C:=sypialniaR.WyjscieOpuszczanie;

sypialniaBalkonR(wejscieSterujace:=inB1,
		ZmiennaPodnoszenieVis:=sypialniaBalkonUpVis,
		ZmiennaOpuszczanieVis:=sypialniaBalkonDnVis,
		ZmiennaLamelkiVis:=sypialniaBalkonLamelkiVis,
		PozycjaLameli:=10,
		CzasOtwarcia:=T#29s,
		CzasZamkniecia:=T#24s,
		MaxCzasDzialania:=T#29s,
		ZamykanieWszystkieVis:=zamykanieWszystkieVis OR opuscPietro,
		OtwieranieWszystkieVis:=otwieranieWszystkieVis OR podniesPietro);
out3D:=sypialniaBalkonR.WyjsciePodnoszenie;
out3E:=sypialniaBalkonR.WyjscieOpuszczanie;
END_PROGRAM

(* POU Rolety2/RoletyFUN, ST *)
FUNCTION_BLOCK RoletyFUN
VAR_INPUT
	WejscieSterujace :BOOL;
	ZmiennaPodnoszenieVis :BOOL;
	ZmiennaOpuszczanieVis :BOOL;
      ZmiennaLamelkiVis :BOOL;
	PozycjaLameli :BYTE;
	CzasOtwarcia: TIME;
	CzasZamkniecia: TIME;
	MaxCzasDzialania :TIME;
	ZamykanieWszystkieVis: BOOL;
	OtwieranieWszystkieVis: BOOL;
END_VAR
VAR_OUTPUT
	WyjsciePodnoszenie :BOOL;
	WyjscieOpuszczanie :BOOL;
	RoletaZamknieta :BOOL;
	RoletaOtwarta: BOOL;
	Pozycja:BYTE;
END_VAR
VAR
	Wejscie1 : Fb_ShortLong:=(uiTS_10tel_s:=1, uiTL_10tel_s:=1, uiT_10tel_s :=5); (* Przycisk w garazu*)
 	Input_B_Roleta4 :BLIND_INPUT;
	czas:SUN_TIME:=(latitude:=51.3,longitude:=17.0);
	Night_B_Roleta4: BLIND_NIGHT:=(NIGHT_POSITION:=0);
    (*Shade_B_Roleta4 :BLIND_SHADE_S:=(HORZ1:=70, HORZ2:=150, SHADE_POS:=150, SHADE_DELAY:=T#60s);*)
    	Control_B_Roleta4 :BLIND_CONTROL_S;
END_VAR
VAR RETAIN PERSISTENT

END_VAR
czas.UTC:=SDT_TO_DATE(DT_TO_SDT(ReadClock.Calendar.UTC));

Wejscie1(xSwitch:=WejscieSterujace);
Input_B_Roleta4(
    S1:=Wejscie1.xShort OR ZmiennaPodnoszenieVis OR OtwieranieWszystkieVis,
    S2:=Wejscie1.xLong OR ZmiennaOpuszczanieVis OR ZamykanieWszystkieVis,
    IN:=ZmiennaLamelkiVis,
    PI:=PozycjaLameli,
    MAX_RUNTIME:= MaxCzasDzialania,
    MANUAL_TIMEOUT:=T#5m,
    MASTER_MODE:=TRUE,
    POS:=Control_B_Roleta4.POS
    );
(*Shade_B_Roleta4(
    UP:=Input_B_Roleta4.QU,
    DN:=Input_B_Roleta4.QD,
    S_IN:=Input_B_Roleta4.STATUS,
    pi:=Input_B_Roleta4.PO,
    ENABLE:=ShadeFlag_B_1S,
    SUN:=SunSignal_1S,
    CX:=ReadClock.Calendar
    );*)

Night_B_Roleta4(
	UP:=Input_B_Roleta4.QU,
	DN:=Input_B_Roleta4.QD,
	S_IN:=Input_B_Roleta4.STATUS,
	PI:=Input_B_Roleta4.PO,
	DTIN:=ReadClock.Calendar.UTC,
	SUNRISE:=ReadClock.Calendar.SUN_RISE,
	SUNSET:=ReadClock.Calendar.SUN_SET(*,
	SUNRISE_OFFSET:=(T#2h-T#4h),
	SUNSET_OFFSET:=T#1h*)
);

Control_B_Roleta4(
   T_UP:= CzasOtwarcia,
   T_DN:= CzasZamkniecia,
    UP:=Night_B_Roleta4.QU,
    DN:=Night_B_Roleta4.QD,
    S_IN:=Night_B_Roleta4.STATUS,
    pi:=Night_B_Roleta4.PO
    );

WyjsciePodnoszenie:=Control_B_Roleta4.MU;
WyjscieOpuszczanie:=Control_B_Roleta4.MD;
Pozycja:=Control_B_Roleta4.POS;


IF (Control_B_Roleta4.POS <= 255 AND Control_B_Roleta4.POS  >= 1) THEN RoletaOtwarta:=TRUE;
ELSE RoletaOtwarta:=FALSE;
END_IF;

IF (Control_B_Roleta4.POS = 0) THEN RoletaZamknieta:=TRUE;
ELSE RoletaZamknieta:=FALSE;
END_IF;


(* Koniec ROLETA4*)
END_FUNCTION_BLOCK

(* POU Rolety2/ReadClock, ST *)
PROGRAM ReadClock
VAR
	Holidays: ARRAY [0..29] OF HOLIDAY_DATA;
	Calendar: CALENDAR := (LATITUDE:=51.3, LONGITUDE:=17.0, OFFSET:=120);
	Calendar_Updater: CALENDAR_CALC := (SPE:=TRUE);
END_VAR
Calendar_Updater(XCAL:=Calendar, HOLIDAYS:=Holidays);
Calendar.Utc:=SysRtcGetTime(TRUE); (*make sure your system runs at UTC time, otherwise - correct it with for example +/- T#2h*)
END_PROGRAM

(* POU Gniazda, ST *)
PROGRAM Gniazda
VAR
END_VAR

END_PROGRAM

(* POU Configuration/MODBUS_CONFIGURATION, ST *)
PROGRAM MODBUS_CONFIGURATION
VAR                                
END_VAR                            
(*                                 
   <?xml version="1.0" encoding="UTF-16" standalone="yes"?>
<network xml_structure_version="1" xml_feature_version="1">
	<generator_settings minRTUTaskCycleTimeMs="5" minEthaskCycleTimeMs="5" ethSlaveMultiplier="0.1" rtuInterfaceMultiplier="0.1" taskGeneration="false"/>
</network>
                              
*)                                 
;                                  
END_PROGRAM

(* POU Rolety2/Rolety4, ST *)
PROGRAM Rolety4
VAR
	Clicker_IN1: Fb_ShortLong := (uiTS_10tel_s:=1, uiTL_10tel_s:=1, uiT_10tel_s :=5);
	ShadeFlag_B_1S: BOOL := FALSE;
	VIS_B_1S1_UP:BOOL:=FALSE;
	VIS_B_1S1_DOWN:BOOL:=FALSE;
END_VAR
VAR RETAIN
	Shade_B_1S1: BLIND_SHADE_S := (HORZ1:=70, HORZ2:=150, SHADE_POS:=150, SHADE_DELAY:=T#60s);
	Input_B_1S1: BLIND_INPUT := (PI:=120, MAX_RUNTIME:=T#25s, MANUAL_TIMEOUT:=t#60m, MASTER_MODE:=TRUE);
	Control_B_1S1: BLIND_CONTROL_S := (T_UP:=T#20s, T_DN:=T#18s);
END_VAR
Clicker_IN1(xSwitch:=input10);
Input_B_1S1(
    S1:=Clicker_IN1.xShort OR VIS_B_1S1_UP,
    S2:=Clicker_IN1.xLong OR VIS_B_1S1_DOWN,
    IN:=VIS_B_1S1_SpecPos,
    POS:=Control_B_1S1.POS
    );
Shade_B_1S1(
    UP:=Input_B_1S1.QU,
    DN:=Input_B_1S1.QD,
    S_IN:=Input_B_1S1.STATUS,
    pi:=Input_B_1S1.PO,
    ENABLE:=ShadeFlag_B_1S,
    SUN:=SunSignal_1S,
    CX:=ReadClock.Calendar
    );
Control_B_1S1(
    UP:=Shade_B_1S1.QU,
    DN:=Shade_B_1S1.QD,
    S_IN:=Shade_B_1S1.STATUS,
    pi:=Shade_B_1S1.PO
    );

output40:=Control_B_1S1.MU;
output41:=Control_B_1S1.MD;
END_PROGRAM

(* POU Satel_RS232/RS232, ST *)
PROGRAM RS232

VAR
    (*interface definitions*)
    CommContext : SERIAL_INTERFACE;
    Init : BOOL;
    Error : BYTE;
    IsOpen : BOOL;
    Send : BOOL:=TRUE; (*send launch, reset on send end*)
    RMessage : typRING_BUFFER; (*received message*)
    Message : POINTER TO BYTE;
    MessageLEN : BYTE;
 
    (*default message to be sent*)
    Message7F : ARRAY [0..6] OF BYTE:=254, 254, 127, 216, 97, 254, 13;
 
    (*variables supervising communication flow*)
    SendEnds : F_TRIG;
    SendStarts : R_TRIG;
    WaitForData : BOOL;
    StopWaiting : TON;
    FrameComplete : BOOL;
    LastRecord : INT; (*stores last reviewed byte*)
    SyncSignal : BOOL:=FALSE;
    EndSignal : BOOL:=FALSE;
 
    (*variables for RMessage analysis*)
    mStart, mEnd : INT;
    crcHigh, crcLow : BYTE;
    RMessageCRC : CRC_Calculate;
    Command : BYTE;
 
    (*variables for preparing message on demand*)
    FoundNewState : BOOL;
    MessageState : typRing_BUFFER;
    MessageStCrc : CRC_Calculate;
    CrcLenExtension : BYTE;
 
    (*variables storing data received from Integra*)
    Sensors : ARRAY[0..55] OF BOOL;
    NewStates : ARRAY[0..39] OF BOOL;
     
    i : BYTE;
END_VAR
SendStarts(CLK:=Send); (*trigger sensing the begin of sending*)
 
IF SendStarts.Q THEN (*if sending starts*)
    (*prepare the variables*)
    FoundNewState:=FALSE;
    i:=0;

    (*checking if there is an unread Integra64 state stored in NewStates ARRAY*)
    WHILE (i<40) AND (NOT FoundNewState) DO
        IF NewStates[i] THEN (*new event found*)
            FoundNewState:=TRUE; (*marker to finish searching*)
            NewStates[i]:=FALSE; (*reset the state in NewState ARRAY*)
            CrcLenExtension:=0;
 
 
            (*preparing new message to be sent*)
            MessageState.Data[0]:=254;
            MessageState.Data[1]:=254;
            MessageState.Data[2]:=i; (*command number=index in the ARRAY*)
            MessageStCrc(m:=ADR(MessageState), start:=2, end:=2); (*calculate CRC*)
            MessageState.Data[3]:=WORD_TO_BYTE(MessageStCrc.hi);
 
            IF MessageStCrc.hi=254 THEN (*if CRC.hi=254 add 240 after it*)
                MessageState.Data[4]:=240;
                CrcLenExtension:=1;
            END_IF;
 
            MessageState.Data[4+CrcLenExtension]:=WORD_TO_BYTE(MessageStCrc.lo);
 
            IF MessageStCrc.lo=254 THEN (*if CRC.lo=254 add 240 after it*)
                MessageState.Data[5+CrcLenExtension]:=240;
                CrcLenExtension:=CrcLenExtension+1;
            END_IF;
 
            MessageState.Data[5+CrcLenExtension]:=254;
            MessageState.Data[6+CrcLenExtension]:=13;
            MessageState.Index:=7+CrcLenExtension;
        END_IF; (*End of IF new event found*)
 
        i:=i+1;
    END_WHILE; (*end of loop for checking NewState ARRAY*)
 
    (*the clue of this IF statement – decide what message to send*)
    IF FoundNewState THEN (*if there is an new state to be red*)
        Message:=ADR(MessageState.Data);
        MessageLen:=INT_TO_BYTE(MessageState.Index);
    ELSE (*otherwise send the standard 7F message*)
        Message:=ADR(Message7F);
        MessageLEN:=7;
    END_IF;
END_IF; (* End of IF Send Start detected*)
 
(*definition of the Communication module*)
CommContext(
    xOPEN_COM_PORT:=TRUE,
    bCOM_PORT_NR:=2,
    cbBAUDRATE:=1920,
    cpPARITY:=0,
    csSTOPBITS:=1,
    cbsBYTESIZE:=8,
    cfFLOW_CONTROL:= 0,
    iBYTES_TO_SEND:=MessageLEN,
    ptSEND_BUFFER:=Message, (*here is where the message pointer goes*)
    xSTART_SEND:=Send,
    utRECEIVE_BUFFER:=RMessage,
    xINIT:= Init,
    bERROR=>Error,
    xCOM_PORT_IS_OPEN=> IsOpen);
 
SendEnds(CLK:= Send); (*trigger sensing the end of sending*)
 
IF SendEnds.Q THEN (*if sending ends…*)
    WaitForData:=TRUE;
END_IF;
 
(* Impulse used to start all over if correct answer is not coming*)
StopWaiting(IN:= WaitForData, PT:=t#1s);
 
IF WaitForData THEN
    (*looking for the bytes 0xFE 0xFE = frame starts
    repeated in next cycles despite finding one 0xFE 0xFE
    in case new sync frame signal comes
    analysis starts from where it ended in the previous cycle*)
 
    WHILE (LastRecord<RMessage.Index-1) DO
        IF RMessage.Data[LastRecord]=254 AND RMessage.Data[LastRecord+1]=254 THEN
            SyncSignal:=TRUE;
            mStart:=LastRecord+2; (*message start marker*)
            LastRecord:=LastRecord+1;
        END_IF;
        LastRecord:=LastRecord+1;
    END_WHILE;
 
    (*reset LastRecord to where the 0xFE 0xFE ended*)
    IF SyncSignal THEN
        LastRecord:=mStart;
    END_IF;
 
    (*looking for bytes 0xFE 0x0D = frame ends*)
    WHILE (LastRecord<RMessage.Index-1) AND SyncSignal DO
        IF RMessage.Data[LastRecord]=254 AND RMessage.Data[LastRecord+1]=13 THEN
            EndSignal:=TRUE;
            mEnd:=LastRecord-1; (*message end marker*)
        END_IF;
        LastRecord:=LastRecord+1;
    END_WHILE;
 
    (*if a complete frame has been received*)
    IF SyncSignal AND EndSignal THEN
        (*check CRC, watch out for 240 bytes - they should be dropped*)
        IF RMessage.Data[mEnd]=240 THEN (*if one of the CRC numbers is 0xF0, drop it*)
            mEnd:=mEnd-1;
        END_IF;
        crcLow:=RMessage.Data[mEnd];
 
        IF RMessage.Data[mEnd-1]=240 THEN (*if one of the CRC numbers is 0xF0, drop it*)
            mEnd:=mEnd-1;
        END_IF;
        crcHigh:=RMessage.Data[mEnd-1];
        mEnd:=mEnd-2;
 
        (*function block for calculating CRC*)
        RMessageCRC(m:=ADR(RMessage), start:=mStart, end:=mEnd);
 
        (*check if CRC is okay*)
        IF RMessageCRC.hi=crcHigh AND RMessageCRC.lo=crcLow THEN
            (*analysis of the received command*)
            Command:=RMessage.Data[mStart];
            CASE Command OF
                (*zones violation*)
                0: IF (mEnd-mStart)>15 THEN (*check for required response length*)
                    FOR i:=0 TO 6 DO
                        Sensors[0+i*8]:=RMessage.Data[mStart+1+i].0;
                        Sensors[1+i*8]:=RMessage.Data[mStart+1+i].1;
                        Sensors[2+i*8]:=RMessage.Data[mStart+1+i].2;
                        Sensors[3+i*8]:=RMessage.Data[mStart+1+i].3;
                        Sensors[4+i*8]:=RMessage.Data[mStart+1+i].4;
                        Sensors[5+i*8]:=RMessage.Data[mStart+1+i].5;
                        Sensors[6+i*8]:=RMessage.Data[mStart+1+i].6;
                        Sensors[7+i*8]:=RMessage.Data[mStart+1+i].7;
                    END_FOR;
                END_IF;
                 
                (*here other commands are to be filled*)
 
                (*list new states*)
                127: IF (mEnd-mStart)>4 THEN (*check for required response length*)
                    FOR i:=0 TO 4 DO
                        NewStates[0+i*8]:=RMessage.Data[mStart+1+i].0;
                        NewStates[1+i*8]:=RMessage.Data[mStart+1+i].1;
                        NewStates[2+i*8]:=RMessage.Data[mStart+1+i].2;
                        NewStates[3+i*8]:=RMessage.Data[mStart+1+i].3;
                        NewStates[4+i*8]:=RMessage.Data[mStart+1+i].4;
                        NewStates[5+i*8]:=RMessage.Data[mStart+1+i].5;
                        NewStates[6+i*8]:=RMessage.Data[mStart+1+i].6;
                        NewStates[7+i*8]:=RMessage.Data[mStart+1+i].7;
                    END_FOR;
                END_IF;
            END_CASE;
        END_IF; (*End of IF CRC OK*)
 
        (*marker to finish waiting and send new message*)
        FrameComplete:=TRUE;
         
    END_IF; (*END of IF a frame has been received*)
END_IF; (*END of IF WaitingForData*)
 
(*if a complete frame has been received or waiting time has passed*)
IF StopWaiting.Q OR FrameComplete THEN
    (*reset all the variables*)
    WaitForData:=FALSE;
    RMessage.Index:=0;
    SyncSignal:=FALSE;
    EndSignal:=FALSE;
    LastRecord:=0;
    mStart:=0;
    mEnd:=0;
    FrameComplete:=FALSE;
    Send:=TRUE;
END_IF;
END_PROGRAM

(* POU Satel_RS232/CRC_Calculate, ST *)
FUNCTION_BLOCK CRC_Calculate
VAR_INPUT
    m : POINTER TO typRing_BUFFER;
    start : INT;
    end :INT;
END_VAR
 
VAR_OUTPUT
    lo : WORD;
    hi : WORD;
    crc : WORD;
END_VAR
 
VAR
    i : INT;
    d : WORD;
    tcrc : WORD;
END_VAR
IF end=0 THEN
    end:=m^.Index;
END_IF;
 
tcrc:=16#147A;
 
FOR i:=start TO end DO
    tcrc:=ROL(tcrc, 1);
    tcrc:=tcrc XOR 16#FFFF;
    tcrc:=tcrc+HEX_HI(in:=tcrc)+m^.Data[i];
END_FOR;
 
crc:=tcrc;
d:=tcrc / 4096;
 
hi:=d*16;
tcrc:=tcrc-d*4096;
d:=tcrc/256;
hi:=hi+d;
 
tcrc:=tcrc-d*256;
d:=tcrc/16;
lo:=d*16;
tcrc:=tcrc-d*16;
lo:=lo+tcrc;
END_FUNCTION_BLOCK

(* POU Satel_RS232/HEX_HI, ST *)
FUNCTION HEX_HI : WORD
VAR_INPUT
    in : WORD;
END_VAR
 
VAR
    div4096 : WORD;
END_VAR
div4096:=in/4096;
HEX_HI:=div4096*16;
in:=in-4096*div4096;
HEX_HI:=HEX_HI+in/256;
END_FUNCTION

(* POU Satel_ETH/Satel, ST *)
PROGRAM Satel
VAR
	czujki:ARRAY[1..64] OF BOOL;
	strefy:ARRAY[1..32] OF BOOL;
	MySatelEthernet : SatelEthernet;

END_VAR
MySatelEthernet(xOpen_Client:=TRUE,IP:='192.168.1.111',Port:=7094);
czujki := MySatelEthernet.czujki;
strefy := MySatelEthernet.strefy;
END_PROGRAM

(* POU Satel_ETH/SatelEthernet, ST *)
FUNCTION_BLOCK SatelEthernet
VAR_INPUT
	xOpen_Client: BOOL;			(* uaktywnij polaczenie do modulu ETHM-1 *)
	IP: STRING;					(* adres IP  modulu ETHM-1 *)
	Port: WORD;					(* port integracji modulu ETHM-1 *)
END_VAR
VAR_OUTPUT
	czujki: ARRAY [1..64] OF BOOL; (* tablica zawierajaca stany czujek od 1 do 64, TRUE - czujka aktywna *)
	strefy: ARRAY [1..32] OF BOOL; (* tablica zawierajaca stany stref od 1 do 32, TRUE - strefa uzbrojona *)
	wyjscia: ARRAY [1..64] OF BOOL; (* tablica zawierajaca stany wyjsc od 1 do 64, TRUE - wyjscie aktywne *)
	xCLIENT_OPEN: BOOL;			(* polaczenie do modulu ETHM-1 aktywne *)
	wSOCKET: WORD;				(* numer wtyczki *)
END_VAR
VAR
	Protocol						: SEL_PROTOCOL 				:= IPPROTO_TCP; (* wybrany protokol transmisji - TCP *)
	ProtocolType					: SEL_TYPE						:= SOCK_STREAM; (* wybrany typ trasmisji - stream *)
	MyEthernetOpen				: ETHERNET_CLIENT_OPEN;
	MyEthernetClose				: ETHERNET_CLIENT_CLOSE;
	MyEthernetWrite				: ETHERNET_WRITE;
	MyEthernetRead				: ETHERNET_READ;
	Read00						: BOOL := TRUE;							(* zadanie wyslania polecenia 00 - odczyt stanu czujek*)
	Read0A						: BOOL := TRUE;							(*zadanie wyslania polecenia 0A - odczyt stanu uzbrojenia alarmu *)
	Read17						: BOOL := TRUE;							(* zadanie wyslania polecenia 00 - odczyt stanu wyjsc*)
	fi: INT;					(* pierwszy  indeks ramki *)
	fin: INT;				(* drugi indeks ramki *)
	buf_len: WORD;		(* dlugosc danych w buforze *)
	znacznik: BYTE := 1;	(* znacznik uzywany do operacji bitowych *)
	pt: POINTER TO ARRAY [1..1500] OF BYTE; (* wskaznik do tablicy - uzywany przy przkazywaniu tablicy do funkcji *)
	frame_rcv: ARRAY [1..1500] OF BYTE;	(* tablica danych odebranych *)
	frame_snd: ARRAY [1..1500] OF BYTE;	(* tablica danych wysylanych *)
	Status: WORD := 0;	(* status transmisji: 0 - inicjalizacja, 1 - sprawdzenie stosu TCP/IP 4 - inicjalizacja otwarcia polaczenia, 5 - oczekiwanie na otwarcie polaczenia, 10 -wyslanie danych do serwera, 20 - oczekiwanie na odbior danych, 30 - interpretacja otrzymanych danych, 40 - zamykanie polaczenia *)
	GetConfig: ETHERNET_GET_NETWORK_CONFIG;
	utERROR: ETH_ERROR;
	closeState: INT;		(* status zamykania polaczenia *)
	Timeout:	TOF_1 := (PT:=T#2s, IN:=TRUE, RST:= FALSE); (* maksymalny czas oczekiwania na odpowiedz ze sterownika *)
END_VAR
IF xOpen_Client THEN

	CASE Status OF
		0:(*Initialize functionblocks*)
			GetConfig(EN:=FALSE );
			GetConfig(EN:=TRUE );
			status:=1;
			utERROR:=0;
			wSocket:=0;
			closeState:=0;
			xCLIENT_OPEN:=FALSE;


		1:(*check ethernet stack*)
			GetConfig(EN:=TRUE );
			IF GetConfig.ENO THEN
				IF GetConfig.IP_ADR<>0 THEN
					status:=4;(*stack initialized*)
				ELSE
					status:=0;(*try again*)
				END_IF
			END_IF


		4:(*open connection*)
			MyEthernetRead(	EN:= 0, SOCKET:=0 ,  DATA:=frame_rcv );
			MyEthernetClose(EN:= 0);
			MyEthernetOpen(EN:=0);

			MyEthernetOpen(EN:=1 , TYP:=ProtocolType	 , PROTO:=Protocol , IP_ADR:= IP_ADDRESS(IP), PORT:=Port );
			status:=5;

		5:(*wait for server response according to client  request to open the connection*)

			MyEthernetOpen(EN:=1, TYP:=ProtocolType, PROTO:=Protocol, IP_ADR:= IP_ADDRESS(IP), PORT:=Port );
			IF  MyEthernetOpen.ENO = 1 THEN
				IF MyEthernetOpen.ERROR = 0 THEN
					Status  := 10; (*socket available*)
					xCLIENT_OPEN:=TRUE;
					wSOCKET	:=MyEthernetOpen.socket;
					MyEthernetWrite(	EN:= 0 , DATA:=frame_snd );
				ELSE
					Status := 0; (*no socket available, try it again *)
				END_IF;
				utERROR:=MyEthernetOpen.ERROR;
			END_IF


		10:(* Write data to server*)

			frame_snd[1]:=16#FE;
			frame_snd[2]:=16#FE;
			IF Read00 THEN
				frame_snd[3]:=16#00;											(* zapytanie o stan czujek *)
			ELSIF Read0A THEN
				frame_snd[3]:=16#0A;											(* zapytanie o stan uzbrojenia alarmu *)
			ELSIF Read17 THEN
				frame_snd[3]:=16#17;											(* zapytanie o stan wyjsc *)
			ELSE
				frame_snd[3]:=16#7F;											(* zapytanie o zmiane stanu *)
			END_IF
			pt:=ADR(frame_snd);
			frame_snd[4]:=WORD_TO_BYTE(SHR(SatelCRC(pt,3,3),8));		(* obliczenie CRC.H *)
			frame_snd[5]:=WORD_TO_BYTE(SatelCRC(pt,3,3));				(* obliczenie CRC.L *)
			frame_snd[6]:=16#FE;
			frame_snd[7]:=16#0D;
			MyEthernetWrite(EN:= 1,SOCKET:= MyEthernetOpen.SOCKET, LEN_IN:=7,DATA:=frame_snd); (* wyslanie ramki *)
			IF MyEthernetWrite.eno THEN
				IF(MyEthernetWrite.ERROR <>0) THEN
					Status:=40;													(* Error writing to the socket, close it *)
				ELSE
					Status:=20; (* Write complete, read data *)
				END_IF;
				utERROR:=MyEthernetWrite.ERROR;
			END_IF
			Timeout (IN := FALSE);


		20:	(* Read data*)

	 		MyEthernetRead(	EN:= 1, SOCKET:=MyEthernetOpen.SOCKET ,  DATA:=frame_rcv );
			MyEthernetRead(	EN:= 0, SOCKET:=0 ,  DATA:=frame_rcv );

			Timeout (IN := FALSE);
			utERROR:=MyEthernetREAD.ERROR;
			IF(MyEthernetRead.ERROR<>0) THEN								(* Error reading the socket, close it *)
				Status:=40;
			ELSIF (MyEthernetRead.LEN_OUT <> 0) THEN  						(* Process the data received via the ethernet port *)
				Timeout(IN := TRUE);
				Status:=30;
			ELSIF NOT Timeout.Q THEN
				Timeout(IN := TRUE);
				Status:=10;														(* uplynal czas oczeiwania na odpowiedz, zerowanie licznika i ponowne wyslanie zapytania *)
			END_IF

		30: (* Process received data *)

			buf_len:=MyEthernetRead.LEN_OUT;
			FOR fi:=3 TO buf_len-4 DO 											(* sprawdzenie, czy bajt odebranej ramki nie zawiera kombinacji FE F0; w takim przypadku wyrzuc F0 i skroc odebrane dane *)
				IF frame_rcv[fi]=16#FE THEN
					IF frame_rcv [fi+1]=16#F0 THEN
						FOR fin:=fi+1 TO buf_len-2 DO
							frame_rcv[fin]:= frame_rcv[fin+1];
						END_FOR
						buf_len:=buf_len-1;
					END_IF;
				END_IF;
			END_FOR;
			pt:=ADR(frame_rcv);													(* przekazanie adresu znacznika danych odebranych - potrzebne do przekazania danych do obliczenia CRC *)
			IF frame_rcv[buf_len-3]=WORD_TO_BYTE(SHR(SatelCRC(pt,3,buf_len-4),8)) AND frame_rcv[buf_len-2]=WORD_TO_BYTE(SatelCRC(pt,3,buf_len-4)) THEN (* sprawdzenie poprawnosci CRC otrzymanych danych *)
				IF frame_rcv[3]=16#7F THEN										(* jesli otrzymano ramke zapytania o zmiane stanu *)
					(*Com7FReceived:=Com7FReceived+1;*)
					IF (frame_rcv[4] AND znacznik) >0 THEN						(* sprawdzenie czy bit 0 pierwszego bajtu danych jest 1, czyli stan czujek ulegl zmianie *)
						Read00:=TRUE;											(* jesli tak, nastepnym razem zapytaj o stan czujek *)
					END_IF;
					IF (frame_rcv[5] AND ROL(znacznik,2)) >0 THEN			(* sprawdzenie czy bit 2 drugiego bajtu danych jest 1, czyli stan stref ulegl zmianie *)
						Read0A:=TRUE;											(* jesli tak, nastepnym razem zapytaj o stan stref*)
					END_IF;
					IF (frame_rcv[6] AND ROL(znacznik,7)) >0 THEN			(* sprawdzenie czy bit 7 trzeciego bajtu danych jest 1, czyli stan wyjsc ulegl zmianie *)
						Read17:=TRUE;											(* jesli tak, nastepnym razem zapytaj o stan wyjsc*)
					END_IF;
				ELSIF frame_rcv[3] = 16#00 THEN								(* jesli otrzymano ramke stanu czujek *)
					(*Com00Received:=Com00Received+1;*)
					znacznik:=1;
					FOR fi:=4 TO buf_len-5 DO									(* dla kazdego bajtu danych *)
						FOR fin:=0 TO 7 DO										(* dla kazdego bitu *)
							IF (SHL(znacznik,fin) AND frame_rcv[fi]) >0 THEN	(* sprawdz czy bit jest 1 *)
								czujki[(fi-4)*8+fin+1]:=TRUE;						(* jesli tak stan czujki = TRUE - aktywna *)
							ELSE
								czujki[(fi-4)*8+fin+1]:=FALSE;						(* jesli nie = FALSE - nieaktywna *)
							END_IF;
						END_FOR;
					END_FOR;
					(*AktCzujek := TRUE;*)
					Read00 := FALSE;;											(* nastepnym razem nie pytaj o czujki *)
				ELSIF frame_rcv[3] = 16#0A THEN
					FOR fi:=4 TO buf_len-5 DO									(* dla kazdego bajtu danych *)
						FOR fin:=0 TO 7 DO										(* dla kazdego bitu *)
							IF (SHL(znacznik,fin) AND frame_rcv[fi]) >0 THEN	(* sprawdz czy bit jest 1 *)
								strefy[(fi-4)*8+fin+1]:=TRUE;						(* jesli tak stan strefy = TRUE - uzbrojona *)
							ELSE
								strefy[(fi-4)*8+fin+1]:=FALSE;						(* jesli nie = FALSE - rozbrojona *)
							END_IF;
						END_FOR;
					END_FOR;
					Read0A := FALSE;											(* nastepnym razem nie pyatj o strefy *)
				ELSIF frame_rcv[3] =16#17 THEN
					FOR fi:=4 TO buf_len-5 DO									(* dla kazdego bajtu danych *)
						FOR fin:=0 TO 7 DO										(* dla kazdego bitu *)
							IF (SHL(znacznik,fin) AND frame_rcv[fi]) >0 THEN	(* sprawdz czy bit jest 1 *)
								wyjscia[(fi-4)*8+fin+1]:=TRUE;						(* jesli tak stan wyjscia = TRUE - aktywne *)
							ELSE
								wyjscia[(fi-4)*8+fin+1]:=FALSE;						(* jesli nie = FALSE - nieaktywne *)
							END_IF;
						END_FOR;
					END_FOR;
					Read17 := FALSE;											(* nastepnym razem nie pyatj o wyjscia *)
				END_IF;
			END_IF;
			Status:=10;															(* przejdz do wysylania danych *)
			MyEthernetWrite(	EN:= 0 , DATA:=frame_snd );						(* przygotuj nadajnik do nadawania *)

		40:	(* Close the client *)

			MyEthernetClose(EN:= 1, SOCKET:= MyEthernetOpen.SOCKET);
			IF MyEthernetClose.eno THEN
				MyEthernetClose(EN:= 0);
				xCLIENT_OPEN:=FALSE;
				Status := 0; (* Try to open the server again *)
			END_IF

	END_CASE;
ELSE
	CASE CloseState OF
	0:
		MyEthernetClose(EN:= 0);
		MyEthernetClose(EN:= 1, SOCKET:= MyEthernetOpen.SOCKET);
		CloseState:=1;
	1:
		MyEthernetClose(EN:= 1, SOCKET:= MyEthernetOpen.SOCKET);
		IF MyEthernetClose.eno THEN
			MyEthernetClose(EN:= 0);
			CloseState:=2;
		END_IF
	2:
		Status := 0;
		utERROR:=0;
		xCLIENT_OPEN:=FALSE;
	END_CASE
END_IF
END_FUNCTION_BLOCK

(* POU Satel_ETH/IP_ADDRESS, ST *)
FUNCTION IP_ADDRESS : DWORD
VAR_INPUT
	IP_ADR	:	STRING;
END_VAR
VAR
	Address 	:	DWORD;
	Value		:	WORD;
	DecimalPos	:	INT;
	Rest		:	STRING;
END_VAR
Address := STRING_TO_WORD(IP_ADR);
IF (Address <= 255) AND (Address >= 0) THEN
	DecimalPos := FIND(IP_ADR,'.');
	IF DecimalPos <> 0 THEN
		Rest := RIGHT(IP_ADR,LEN(IP_ADR) - DecimalPos);
		Value := STRING_TO_WORD(Rest);
		IF (Value <= 255) AND (Value >= 0) THEN
			Address := (Address * 16#0100) + Value;

			DecimalPos := FIND(Rest,'.');
			IF DecimalPos <> 0 THEN
				Rest := RIGHT(IP_ADR,LEN(Rest) - DecimalPos);
				Value := STRING_TO_WORD(Rest);
				IF (Value <= 255) AND (Value >= 0) THEN
					Address := (Address * 16#0100) + Value;

					DecimalPos := FIND(Rest,'.');
					IF DecimalPos <> 0 THEN
						Rest := RIGHT(IP_ADR,LEN(Rest) - DecimalPos);
						Value := STRING_TO_WORD(Rest);
						IF (Value <= 255) AND (Value >= 0) THEN
							Address := (Address * 16#0100) + Value;
						ELSE
							Address := 0;
						END_IF
					ELSE
						Address := 0;
					END_IF
				ELSE
					Address := 0;
				END_IF
			ELSE
				Address := 0;
			END_IF
		ELSE
			Address := 0;
		END_IF
	ELSE
		Address := 0;
	END_IF
ELSE
	Address := 0;
END_IF
IP_ADDRESS := Address;
END_FUNCTION

(* POU Satel_ETH/SatelCRC, ST *)
FUNCTION SatelCRC : WORD
VAR_INPUT
	pt: POINTER TO ARRAY [1..1500] OF BYTE;
	start_pos: INT;
	end_pos: INT;
END_VAR
VAR
	i: INT :=0;
END_VAR
SatelCRC:= 16#147A;
FOR i:=start_pos TO end_pos DO
	SatelCRC:= ROL(SatelCRC,1);
	SatelCRC:= SatelCRC XOR 16#FFFF;
	SatelCRC:= SatelCRC + SHR(SatelCRC,8) + pt^[i];
END_FOR
END_FUNCTION

(* POU Swiatlo2/Zewnetrzne, ST *)
PROGRAM Zewnetrzne
VAR
	wlaczWszystkieSw: BOOL:=FALSE;
	wylaczWszystkieSw: BOOL:=FALSE;
END_VAR

END_PROGRAM

(* Visualisation test
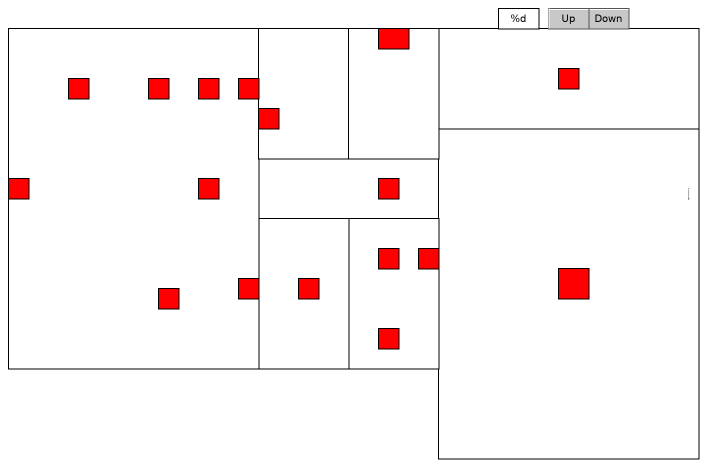
rectangle at (600,340)-(631,371): alarm colour if GarazKotlownia.swGaraz.xActuator; taps GarazKotlownia.visGaraz
rectangle at (420,100)-(451,121): alarm colour if PLC_PRG.swGaraz.xActuator; taps PLC_PRG.visGaraz
rectangle at (460,320)-(481,341): alarm colour if PLC_PRG.swGaraz.xActuator; taps PLC_PRG.visGaraz
rectangle at (420,320)-(441,341): alarm colour if LazienkaParter.swMalaLazienka.xActuator; taps LazienkaParter.visMalaLazienka
rectangle at (420,400)-(441,421): alarm colour if PLC_PRG.swGaraz.xActuator; taps PLC_PRG.visGaraz
rectangle at (340,350)-(361,371): alarm colour if WiatrolapSpizarnia.swWiatrolap.xActuator; taps WiatrolapSpizarnia.visWiatrolap
rectangle at (420,250)-(441,271): alarm colour if PLC_PRG.swGaraz.xActuator; taps PLC_PRG.visGaraz
rectangle at (240,250)-(261,271): alarm colour if PLC_PRG.swGaraz.xActuator; taps PLC_PRG.visGaraz
rectangle at (200,360)-(221,381): alarm colour if Salon.swSalonCentralne.xActuator; taps PLC_PRG.visGaraz
rectangle at (50,250)-(71,271): alarm colour if Salon.swSalonSciana.xActuator; taps Salon.visSalonSciana
rectangle at (240,150)-(261,171): alarm colour if PLC_PRG.swGaraz.xActuator; taps PLC_PRG.visGaraz
rectangle at (190,150)-(211,171): alarm colour if KuchniaJadalnia.swBlat.xActuator; taps KuchniaJadalnia.visBlat
rectangle at (110,150)-(131,171): alarm colour if KuchniaJadalnia.swJadalnia.xActuator; taps KuchniaJadalnia.visJadalnia
rectangle at (600,140)-(621,161): alarm colour if GarazKotlownia.swKotlownia.xActuator; taps GarazKotlownia.visKotlownia
rectangle at (300,180)-(321,201): alarm colour if PLC_PRG.swGaraz.xActuator; taps PLC_PRG.visGaraz
rectangle at (280,150)-(301,171): alarm colour if PLC_PRG.swGaraz.xActuator; taps PLC_PRG.visGaraz
rectangle at (280,350)-(301,371): alarm colour if PLC_PRG.swGaraz.xActuator; taps PLC_PRG.visGaraz
button at (630,80)-(671,101): text "Down"; taps RoletaKotlownia.VIS_Blind_1_DN
button at (590,80)-(631,101): text "Up"; taps RoletaKotlownia.VIS_Blind_1_UP
rectangle at (540,80)-(581,101): text "%d"; shows RoletaKotlownia.Input_Blind_1.PO
8 more shapes without text or variables
4 elements of other kinds (tables, trends, ...) not read
*)
